// TIA Portal V20 export
DATA_BLOCK "instFB_AutoCtrl_ABCDE"   // DB
TITLE = ABCDE Auto Cycle instance DB
{ S7_Optimized_Access := 'TRUE' }
// iDB for FB_AutoCtrl_ABCDE — Wang Shuo 4-REGION ABCDE 6-state machine + MC_MoveLinearAbsolute
// stored: InstanceOfName FB_AutoCtrl_ABCDE, InstanceOfType FB
"FB_AutoCtrl_ABCDE"
BEGIN
END_DATA_BLOCK
